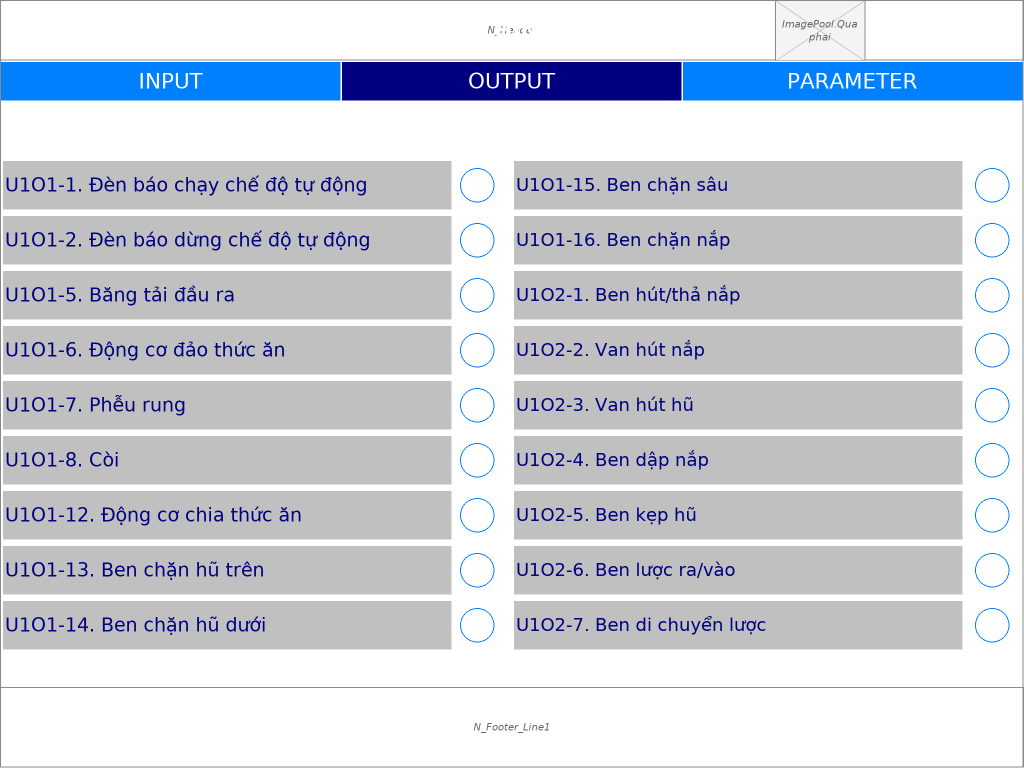
VISUALIZATION N_PLC_O1  // 1024x768
    Frame (0,687 1024x80)
        shows N_Footer_Line1()
    Frame (0,0 1024x60)
        shows N_Header()
    Textfield (353,5 400x50), "MÀN HÌNH IO LINE 1"
    Image (775,0 90x61), image: ImagePool.Qua phai
        OnMouseClick: change screen: N_PLC_O2
    Rectangle (2,160 450x50), "U1O1-1. Đèn báo chạy chế độ tự động"
    Rectangle (2,215 450x50), "U1O1-2. Đèn báo dừng chế độ tự động"
    Rectangle (2,270 450x50), "U1O1-5. Băng tải đầu ra"
    Ellipse (460,168 34x34), colour toggle: GVL_IO.bLight_Running, input disabled if: true
    Ellipse (460,223 34x34), colour toggle: GVL_IO.bLight_Stop, input disabled if: true
    Rectangle (2,325 450x50), "U1O1-6. Động cơ đảo thức ăn"
    Rectangle (2,380 450x50), "U1O1-7. Phễu rung"
    Rectangle (2,435 450x50), "U1O1-8. Còi"
    Rectangle (2,490 450x50), "U1O1-12. Động cơ chia thức ăn"
    Rectangle (2,545 450x50), "U1O1-13. Ben chặn hũ trên"
    Rectangle (2,600 450x50), "U1O1-14. Ben chặn hũ dưới"
    Rectangle (513,160 450x50), "U1O1-15. Ben chặn sâu"
    Rectangle (513,215 450x50), "U1O1-16. Ben chặn nắp"
    Ellipse (460,278 34x34), colour toggle: PR_Conveyor_Out.fb_Conveyor.fbInverter.bVFD, input disabled if: true
    Ellipse (460,333 34x34), colour toggle: PR_Line01.fb_FoodMixer.fbInverter.bVFD, input disabled if: true
    Ellipse (460,388 34x34), colour toggle: PR_Line01.fb_WormWeight.fbInverter.bVFD, input disabled if: true
    Ellipse (460,443 34x34), colour toggle: GVL_IO.bSirens, input disabled if: true
    Ellipse (460,498 34x34), colour toggle: PR_Line01.fb_FoodWeight.fbDriver.bVFD, input disabled if: true
    Ellipse (460,553 34x34), colour toggle: PR_Line01.fb_CupSupply.fbCylinder_Up.bMoveExtend, input disabled if: true
    Ellipse (460,608 34x34), colour toggle: PR_Line01.fb_CupSupply.fbCylinder_Dw.bMoveRetract, input disabled if: true
    Ellipse (975,168 34x34), colour toggle: PR_Line02.fb_WormWeight.fbCylinder.bMoveRetract, input disabled if: true
    Ellipse (975,223 34x34), colour toggle: PR_Line01.fb_LidSupply.fbCylinder_LidStopper.bMoveRetract, input disabled if: true
    Rectangle (513,270 450x50), "U1O2-1. Ben hút/thả nắp"
    Ellipse (975,278 34x34), colour toggle: PR_Line02.fb_LidSupply.fbCylinder_Suction.bMoveExtend, input disabled if: true
    Rectangle (513,325 450x50), "U1O2-2. Van hút nắp"
    Rectangle (513,380 450x50), "U1O2-3. Van hút hũ"
    Rectangle (513,435 450x50), "U1O2-4. Ben dập nắp"
    Rectangle (513,490 450x50), "U1O2-5. Ben kẹp hũ"
    Rectangle (513,545 450x50), "U1O2-6. Ben lược ra/vào"
    Rectangle (513,600 450x50), "U1O2-7. Ben di chuyển lược"
    Ellipse (975,333 34x34), colour toggle: PR_Line02.fb_LidSupply.fbLidSuctionValve.bSuck, input disabled if: true
    Ellipse (975,388 34x34), colour toggle: PR_Line02.fb_LidSupply.fbCupSuctionValve.bSuck, input disabled if: true
    Ellipse (975,443 34x34), colour toggle: PR_Line02.fb_LidClose.fbCylinder_LidClose.bMoveExtend, input disabled if: true
    Ellipse (975,498 34x34), colour toggle: PR_Line01.fb_Transfer.fbCylinder_Clip.bMoveRetract, input disabled if: true
    Ellipse (975,553 34x34), colour toggle: PR_Line01.fb_Transfer.fbCylinder_Comb.bMoveExtend, input disabled if: true
    Ellipse (975,608 34x34), colour toggle: PR_Line01.fb_Transfer.fbCylinder_Move_Comb.bMoveExtend, input disabled if: true
    Rectangle (0,61 341x40), "INPUT"
        OnMouseClick: change screen: N_PLC_I1
    Rectangle (341,61 341x40), "OUTPUT"
        OnMouseClick: change screen: N_PLC_O1
    Rectangle (682,61 341x40), "PARAMETER"
        OnMouseClick: change screen: N_Parameter_1
END_VISUALIZATION

(* stored: Version 1.1.0.1, ProductVersion 3.1.4024.12
   Visu N_PLC_O1: Id {88840a11-3df8-4a4c-b04e-c3f9c1a2ef70} *)
